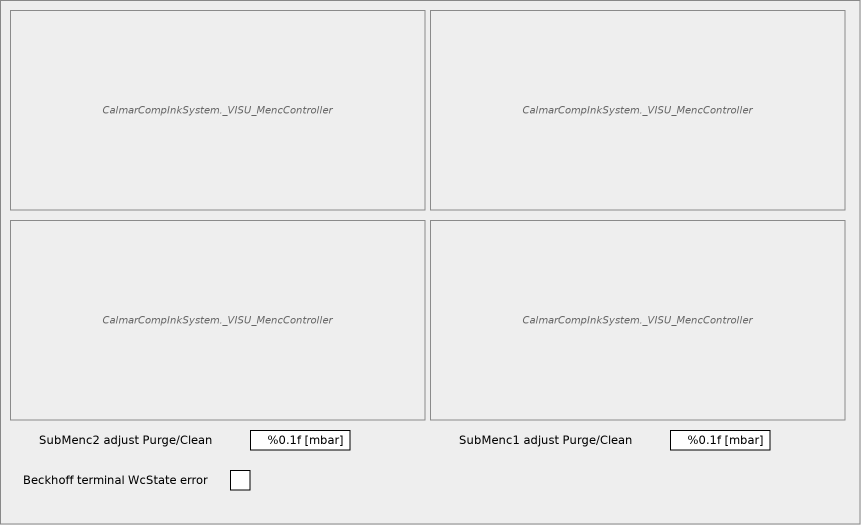
VISUALIZATION VISU_VACUUM  // 861x525
    Rectangle (0,0 861x525)
    RoundedRectangle (230,470 20x20), colour toggle: PRG_INK.bI_InkLevel1WcState
    Rectangle (20,470 200x20), "Beckhoff terminal WcState error"
    Frame (10,10 415x200)
        shows CalmarCompInkSystem._VISU_MencController(m_Inst_Fb := PRG_INK.fb_DgasMencContr[1])
    Frame (430,10 415x200)
        shows CalmarCompInkSystem._VISU_MencController(m_Inst_Fb := PRG_INK.fb_MeniscusMencContr[1])
    Frame (430,220 415x200)
        shows CalmarCompInkSystem._VISU_MencController(m_Inst_Fb := PRG_INK.fb_MeniscusMencContr[2])
    Frame (10,220 415x200)
        shows CalmarCompInkSystem._VISU_MencController(m_Inst_Fb := PRG_INK.fb_MeniscusMencContr[3])
    Rectangle (36,430 209x20), "SubMenc2 adjust Purge/Clean"
    Rectangle (250,430 100x20), "%0.1f [mbar]", text variable: PRG_INK.fR_SubMencSetAdjustWhilePurgeClean[2]
        OnMouseClick: write the text variable via Default
    Rectangle (456,430 209x20), "SubMenc1 adjust Purge/Clean"
    Rectangle (670,430 100x20), "%0.1f [mbar]", text variable: PRG_INK.fR_SubMencSetAdjustWhilePurgeClean[1]
        OnMouseClick: write the text variable via Default
END_VISUALIZATION

(* stored: Version 1.1.0.1, ProductVersion 3.1.4024.9
   Visu VISU_VACUUM: Id {04fa1b6c-d19a-4d13-aa84-22bb3e8e2dbb} *)
